TYPE HLSInputData :
STRUCT
	//In
	iIn : INT;
END_STRUCT
END_TYPE

(* stored: Version 1.1.0.1, ProductVersion 3.1.4024.12
   DUT HLSInputData: Id {b7ee233d-fa98-4915-a0bd-2c662de7786f} *)
